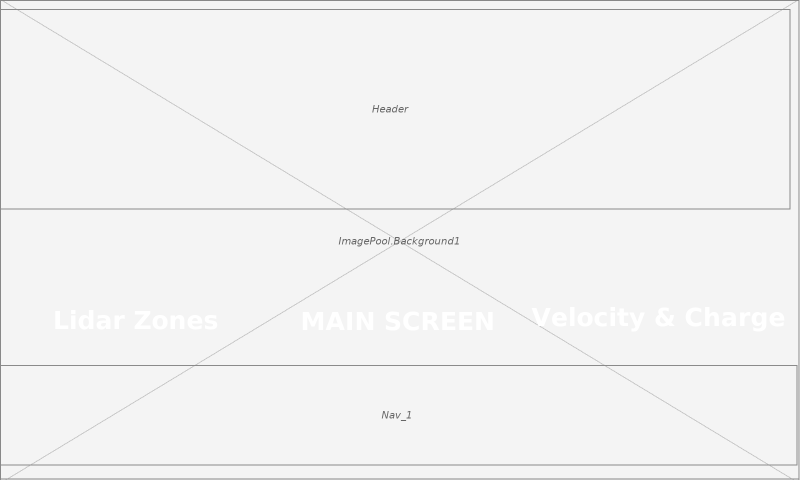
VISUALIZATION MainScreen  // 800x480
    Image (0,-1 799x484), image: ImagePool.Background1
    Frame (-10,9 800x200)
        shows Header()
    Frame (-3,365 800x100)
        shows Nav_1()
    RoundedRectangle (291,289 214x64), "MAIN SCREEN"
    RoundedRectangle (531,285 255x64), "Velocity & Charge"
    RoundedRectangle (29,288 214x64), "Lidar Zones"
END_VISUALIZATION

(* stored: Version 1.1.0.1, ProductVersion 3.1.4024.12
   Visu MainScreen: Id {c793f115-216e-4dc9-b614-f066b4074ef2} *)
